TYPE ST_CFG_TransferCC :
(**************************************************************************************
 * 	Application		:	BoxControl Framework
 *	Revision		:	$Revision: 417092 $
 *	Revision date	:	$Date: 2018-11-14 12:58:58 +0100 (Mi., 14 Nov 2018) $
 *	Last changed by	:	$Author: q8aberh $
 *	URL				:	$URL: http://almscdc.swisslog.com/repo/SWPD/Development/ProMove/02_Controls/ProBox/03_Implementation/01_DevelopmentProject/01_Software/ProBox_COE/ProBox_DevProj_v1.0/PLC_1/20_Product/10_App/12_E_Functions/11_ProBox/21_LowLiftUnit/10_App/01_DUTs/ST_CFG_L $
 *
 *	Purpose			:	Specific configuration for DummyFunction
 *
 * ------------------------------------------------------------------------------------
 *	Copyright Swisslog [IP AG], Switzerland. All rights reserved.
 * 
 * ------------------------------------------------------------------------------------
 *	
 * 	Revision History: 
 *
 * 	VERSION			DATE			INITIALS			DESCRIPTION
 *	0.1				01.01.2001		swl					Example
 *
 **************************************************************************************)	
STRUCT
	HW_InputInverted 				: ST_HW_InputsTransferCC;
	TimeoutValueMotor				: TIME; // Timeout value for Motor
	ReleaseBreakTime				: TIME; // Time before activaring break after running sideshift motor
	HomePosFree						: E_Positions_HorizontalControl; // Homeposition lift when zone free
	HomePosOccupied					: E_Positions_HorizontalControl; // Homeposition lift when zone occupied

END_STRUCT
END_TYPE

(* stored: Version 1.1.0.1, ProductVersion 3.1.4024.9
   DUT ST_CFG_TransferCC: Id {8ffeb045-23ba-4832-988d-762907b8dfa4} *)
